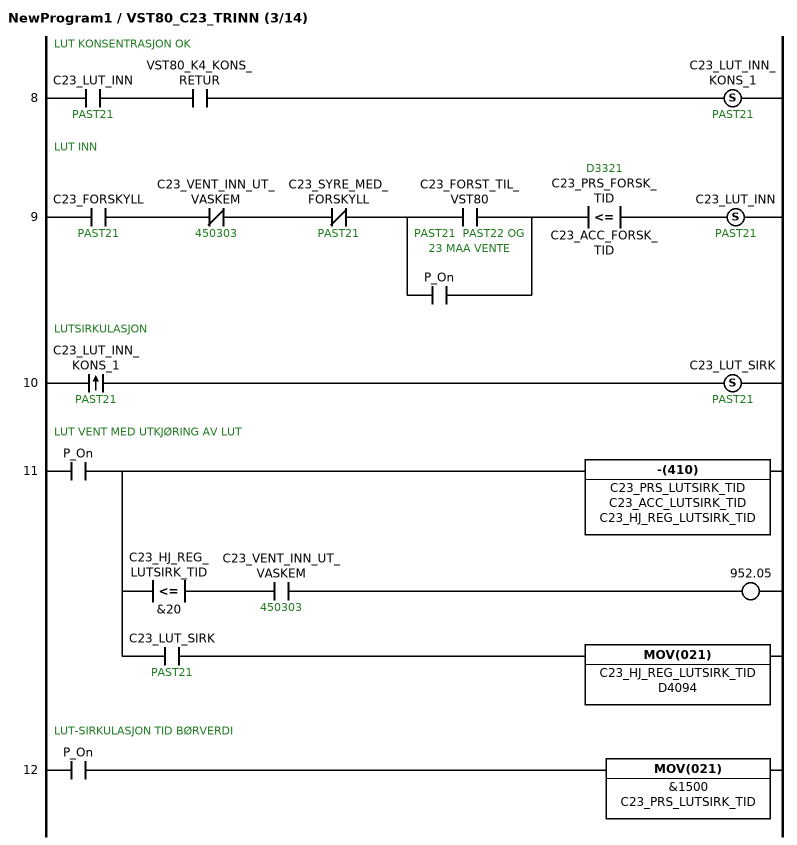
; [picture p408: NewProgram1 / VST80_C23_TRINN, rungs 8-12]
; rung 8: LUT KONSENTRASJON OK
LD C23_LUT_INN  ; PAST21
AND VST80_K4_KONS_RETUR
SET C23_LUT_INN_KONS_1  ; PAST21
; rung 9: LUT INN
LD C23_FORSKYLL  ; PAST21
ANDNOT C23_VENT_INN_UT_VASKEM  ; 450303
ANDNOT C23_SYRE_MED_FORSKYLL  ; PAST21
LD C23_FORST_TIL_VST80  ; PAST21  PAST22 OG 23 MAA VENTE
OR P_On
ANDLD
AND<=(315) C23_PRS_FORSK_TID C23_ACC_FORSK_TID  ; D3321
SET C23_LUT_INN  ; PAST21
; rung 10: LUTSIRKULASJON
@LD C23_LUT_INN_KONS_1  ; PAST21
SET C23_LUT_SIRK  ; PAST21
; rung 11: LUT VENT MED UTKJØRING AV LUT
LD P_On
OUT TR0
-(410) C23_PRS_LUTSIRK_TID C23_ACC_LUTSIRK_TID C23_HJ_REG_LUTSIRK_TID
AND<=(315) C23_HJ_REG_LUTSIRK_TID &20
AND C23_VENT_INN_UT_VASKEM  ; 450303
OUT 952.05
LD TR0
AND C23_LUT_SIRK  ; PAST21
MOV(021) C23_HJ_REG_LUTSIRK_TID D4094
; rung 12: LUT-SIRKULASJON TID BØRVERDI
LD P_On
MOV(021) &1500 C23_PRS_LUTSIRK_TID

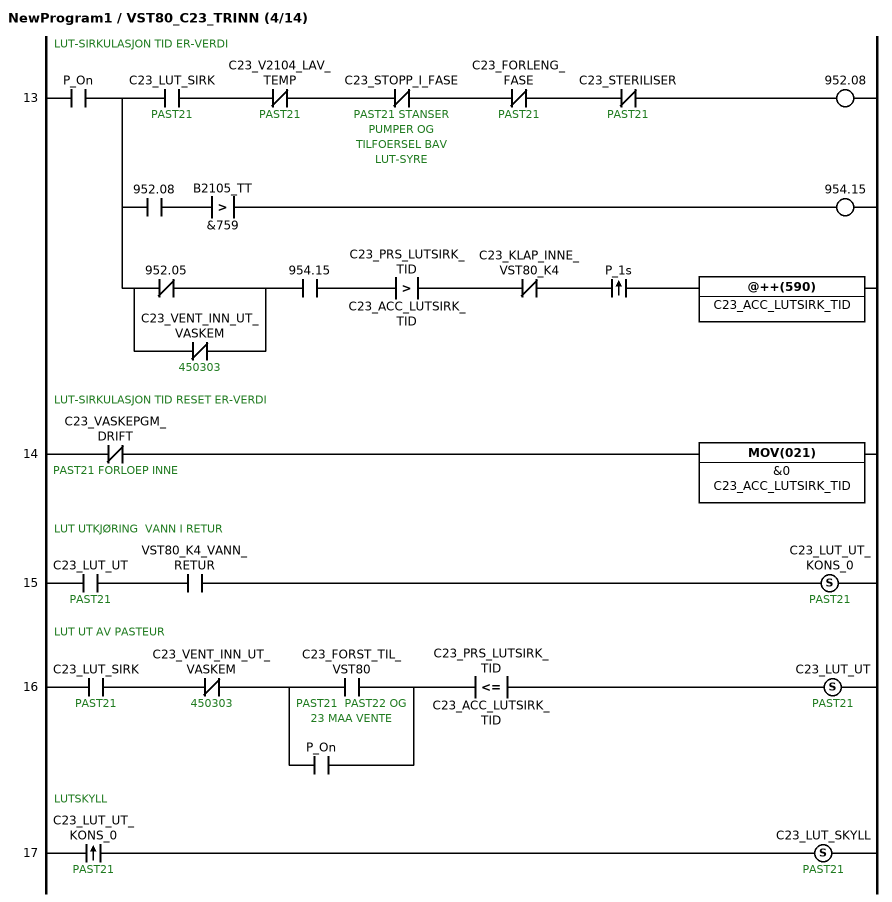
; rung 13: LUT-SIRKULASJON TID ER-VERDI
LD P_On
OUT TR0
AND C23_LUT_SIRK  ; PAST21
ANDNOT C23_V2104_LAV_TEMP  ; PAST21
ANDNOT C23_STOPP_I_FASE  ; PAST21 STANSER PUMPER OG TILFOERSEL BAV LUT-SYRE
ANDNOT C23_FORLENG_FASE  ; PAST21
ANDNOT C23_STERILISER  ; PAST21
OUT 952.08
LD TR0
AND 952.08
AND>(320) B2105_TT &759
OUT 954.15
LD TR0
LDNOT 952.05
ORNOT C23_VENT_INN_UT_VASKEM  ; 450303
ANDLD
AND 954.15
AND>(320) C23_PRS_LUTSIRK_TID C23_ACC_LUTSIRK_TID
ANDNOT C23_KLAP_INNE_VST80_K4
@AND P_1s
@++(590) C23_ACC_LUTSIRK_TID
; rung 14: LUT-SIRKULASJON TID RESET ER-VERDI
LDNOT C23_VASKEPGM_DRIFT  ; PAST21 FORLOEP INNE
MOV(021) &0 C23_ACC_LUTSIRK_TID
; rung 15: LUT UTKJØRING  VANN I RETUR
LD C23_LUT_UT  ; PAST21
AND VST80_K4_VANN_RETUR
SET C23_LUT_UT_KONS_0  ; PAST21
; rung 16: LUT UT AV PASTEUR
LD C23_LUT_SIRK  ; PAST21
ANDNOT C23_VENT_INN_UT_VASKEM  ; 450303
LD C23_FORST_TIL_VST80  ; PAST21  PAST22 OG 23 MAA VENTE
OR P_On
ANDLD
AND<=(315) C23_PRS_LUTSIRK_TID C23_ACC_LUTSIRK_TID
SET C23_LUT_UT  ; PAST21
; rung 17: LUTSKYLL
@LD C23_LUT_UT_KONS_0  ; PAST21
SET C23_LUT_SKYLL  ; PAST21

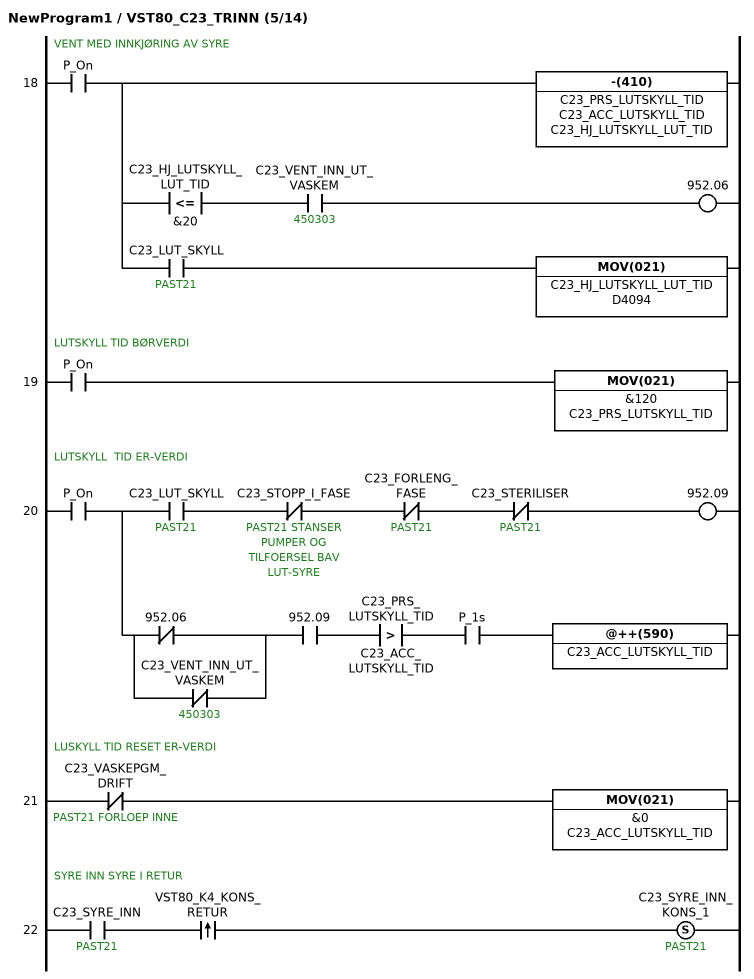
; rung 18: VENT MED INNKJØRING AV SYRE
LD P_On
OUT TR0
-(410) C23_PRS_LUTSKYLL_TID C23_ACC_LUTSKYLL_TID C23_HJ_LUTSKYLL_LUT_TID
AND<=(315) C23_HJ_LUTSKYLL_LUT_TID &20
AND C23_VENT_INN_UT_VASKEM  ; 450303
OUT 952.06
LD TR0
AND C23_LUT_SKYLL  ; PAST21
MOV(021) C23_HJ_LUTSKYLL_LUT_TID D4094
; rung 19: LUTSKYLL TID BØRVERDI
LD P_On
MOV(021) &120 C23_PRS_LUTSKYLL_TID
; rung 20: LUTSKYLL  TID ER-VERDI
LD P_On
OUT TR0
AND C23_LUT_SKYLL  ; PAST21
ANDNOT C23_STOPP_I_FASE  ; PAST21 STANSER PUMPER OG TILFOERSEL BAV LUT-SYRE
ANDNOT C23_FORLENG_FASE  ; PAST21
ANDNOT C23_STERILISER  ; PAST21
OUT 952.09
LD TR0
LDNOT 952.06
ORNOT C23_VENT_INN_UT_VASKEM  ; 450303
ANDLD
AND 952.09
AND>(320) C23_PRS_LUTSKYLL_TID C23_ACC_LUTSKYLL_TID
AND P_1s
@++(590) C23_ACC_LUTSKYLL_TID
; rung 21: LUSKYLL TID RESET ER-VERDI
LDNOT C23_VASKEPGM_DRIFT  ; PAST21 FORLOEP INNE
MOV(021) &0 C23_ACC_LUTSKYLL_TID
; rung 22: SYRE INN SYRE I RETUR
LD C23_SYRE_INN  ; PAST21
@AND VST80_K4_KONS_RETUR
SET C23_SYRE_INN_KONS_1  ; PAST21

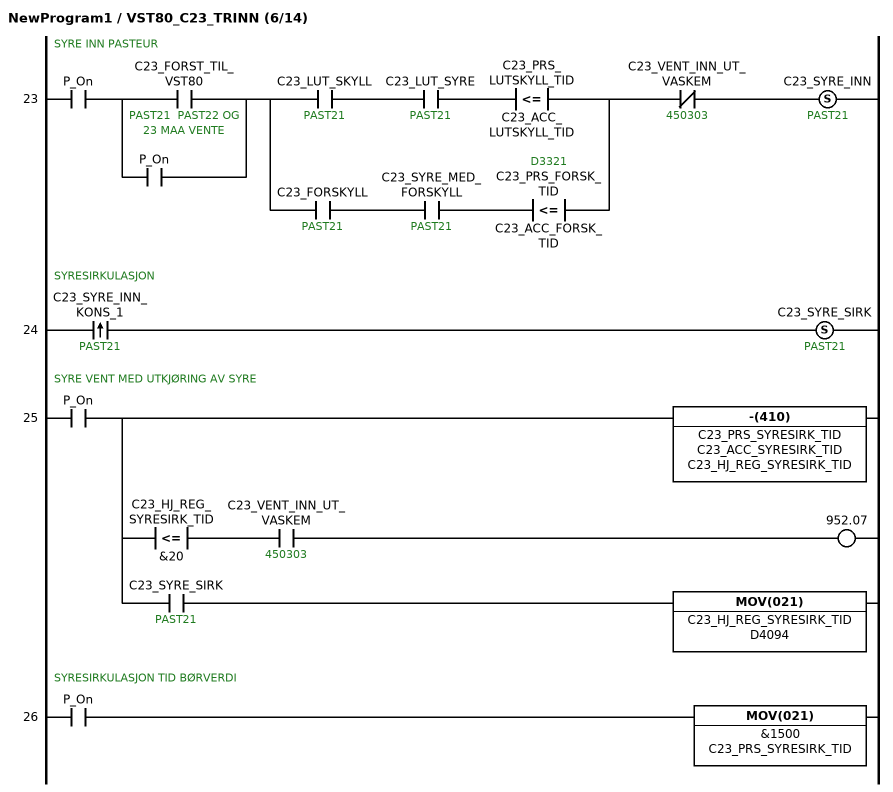
; rung 23: SYRE INN PASTEUR
LD P_On
LD C23_FORST_TIL_VST80  ; PAST21  PAST22 OG 23 MAA VENTE
OR P_On
ANDLD
LD C23_LUT_SKYLL  ; PAST21
AND C23_LUT_SYRE  ; PAST21
AND<=(315) C23_PRS_LUTSKYLL_TID C23_ACC_LUTSKYLL_TID
LD C23_FORSKYLL  ; PAST21
AND C23_SYRE_MED_FORSKYLL  ; PAST21
AND<=(315) C23_PRS_FORSK_TID C23_ACC_FORSK_TID  ; D3321
ORLD
ANDLD
ANDNOT C23_VENT_INN_UT_VASKEM  ; 450303
SET C23_SYRE_INN  ; PAST21
; rung 24: SYRESIRKULASJON
@LD C23_SYRE_INN_KONS_1  ; PAST21
SET C23_SYRE_SIRK  ; PAST21
; rung 25: SYRE VENT MED UTKJØRING AV SYRE
LD P_On
OUT TR0
-(410) C23_PRS_SYRESIRK_TID C23_ACC_SYRESIRK_TID C23_HJ_REG_SYRESIRK_TID
AND<=(315) C23_HJ_REG_SYRESIRK_TID &20
AND C23_VENT_INN_UT_VASKEM  ; 450303
OUT 952.07
LD TR0
AND C23_SYRE_SIRK  ; PAST21
MOV(021) C23_HJ_REG_SYRESIRK_TID D4094
; rung 26: SYRESIRKULASJON TID BØRVERDI
LD P_On
MOV(021) &1500 C23_PRS_SYRESIRK_TID

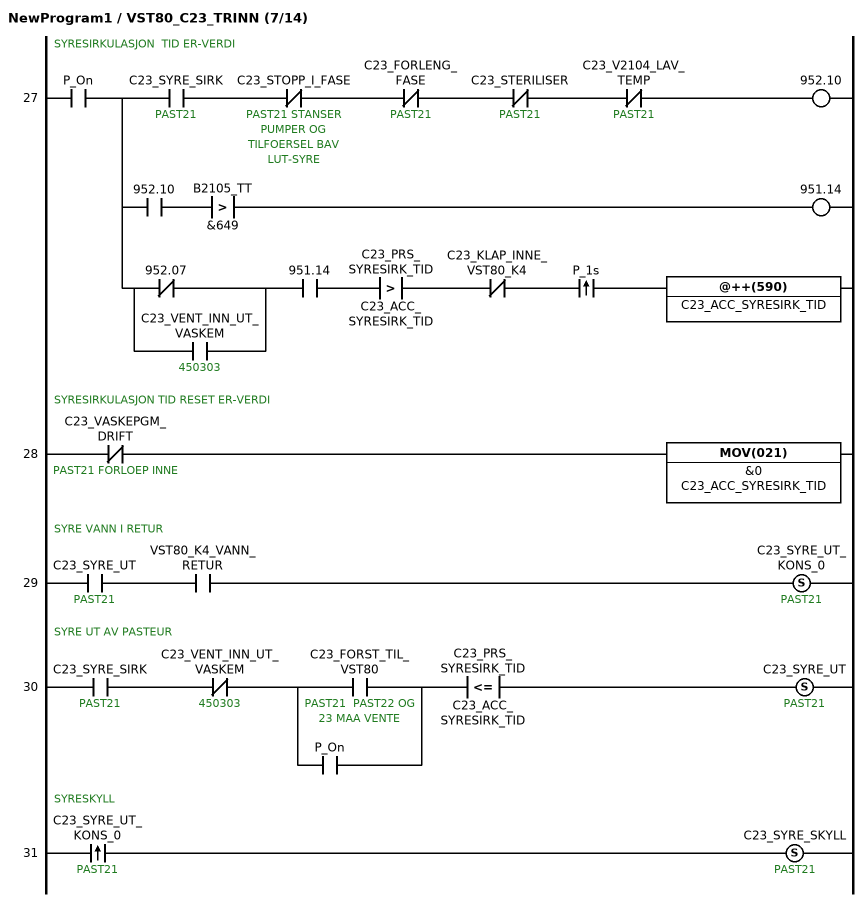
; rung 27: SYRESIRKULASJON  TID ER-VERDI
LD P_On
OUT TR0
AND C23_SYRE_SIRK  ; PAST21
ANDNOT C23_STOPP_I_FASE  ; PAST21 STANSER PUMPER OG TILFOERSEL BAV LUT-SYRE
ANDNOT C23_FORLENG_FASE  ; PAST21
ANDNOT C23_STERILISER  ; PAST21
ANDNOT C23_V2104_LAV_TEMP  ; PAST21
OUT 952.10
LD TR0
AND 952.10
AND>(320) B2105_TT &649
OUT 951.14
LD TR0
LDNOT 952.07
OR C23_VENT_INN_UT_VASKEM  ; 450303
ANDLD
AND 951.14
AND>(320) C23_PRS_SYRESIRK_TID C23_ACC_SYRESIRK_TID
ANDNOT C23_KLAP_INNE_VST80_K4
@AND P_1s
@++(590) C23_ACC_SYRESIRK_TID
; rung 28: SYRESIRKULASJON TID RESET ER-VERDI
LDNOT C23_VASKEPGM_DRIFT  ; PAST21 FORLOEP INNE
MOV(021) &0 C23_ACC_SYRESIRK_TID
; rung 29: SYRE VANN I RETUR
LD C23_SYRE_UT  ; PAST21
AND VST80_K4_VANN_RETUR
SET C23_SYRE_UT_KONS_0  ; PAST21
; rung 30: SYRE UT AV PASTEUR
LD C23_SYRE_SIRK  ; PAST21
ANDNOT C23_VENT_INN_UT_VASKEM  ; 450303
LD C23_FORST_TIL_VST80  ; PAST21  PAST22 OG 23 MAA VENTE
OR P_On
ANDLD
AND<=(315) C23_PRS_SYRESIRK_TID C23_ACC_SYRESIRK_TID
SET C23_SYRE_UT  ; PAST21
; rung 31: SYRESKYLL
@LD C23_SYRE_UT_KONS_0  ; PAST21
SET C23_SYRE_SKYLL  ; PAST21

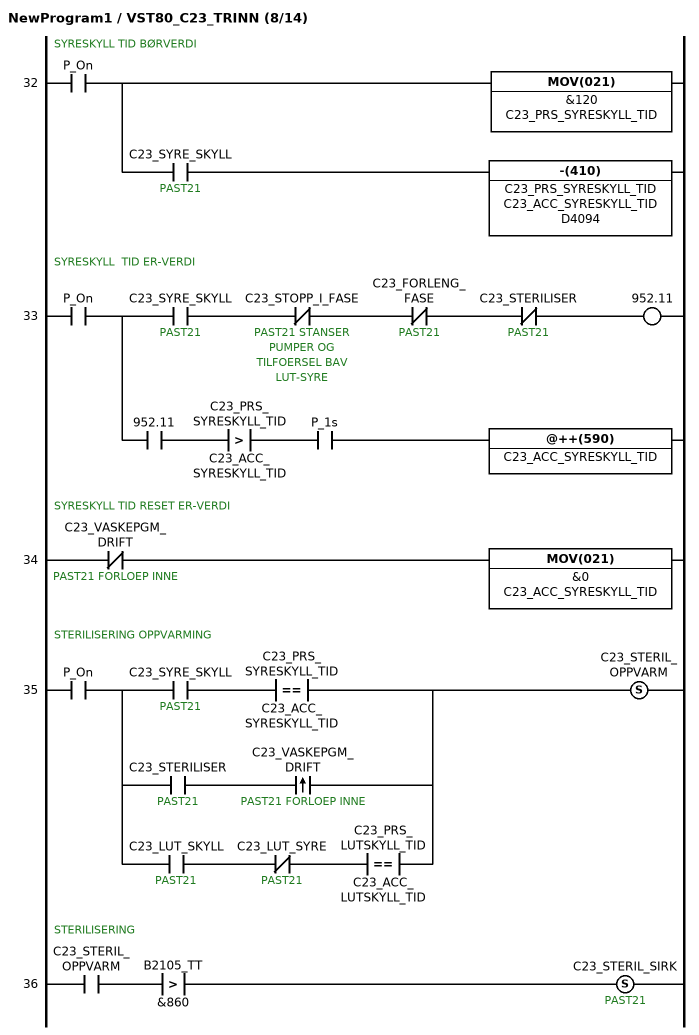
; rung 32: SYRESKYLL TID BØRVERDI
LD P_On
MOV(021) &120 C23_PRS_SYRESKYLL_TID
AND C23_SYRE_SKYLL  ; PAST21
-(410) C23_PRS_SYRESKYLL_TID C23_ACC_SYRESKYLL_TID D4094
; rung 33: SYRESKYLL  TID ER-VERDI
LD P_On
OUT TR0
AND C23_SYRE_SKYLL  ; PAST21
ANDNOT C23_STOPP_I_FASE  ; PAST21 STANSER PUMPER OG TILFOERSEL BAV LUT-SYRE
ANDNOT C23_FORLENG_FASE  ; PAST21
ANDNOT C23_STERILISER  ; PAST21
OUT 952.11
LD TR0
AND 952.11
AND>(320) C23_PRS_SYRESKYLL_TID C23_ACC_SYRESKYLL_TID
AND P_1s
@++(590) C23_ACC_SYRESKYLL_TID
; rung 34: SYRESKYLL TID RESET ER-VERDI
LDNOT C23_VASKEPGM_DRIFT  ; PAST21 FORLOEP INNE
MOV(021) &0 C23_ACC_SYRESKYLL_TID
; rung 35: STERILISERING OPPVARMING
LD P_On
LD C23_SYRE_SKYLL  ; PAST21
AND=(300) C23_PRS_SYRESKYLL_TID C23_ACC_SYRESKYLL_TID
LD C23_STERILISER  ; PAST21
@AND C23_VASKEPGM_DRIFT  ; PAST21 FORLOEP INNE
ORLD
LD C23_LUT_SKYLL  ; PAST21
ANDNOT C23_LUT_SYRE  ; PAST21
AND=(300) C23_PRS_LUTSKYLL_TID C23_ACC_LUTSKYLL_TID
ORLD
ANDLD
SET C23_STERIL_OPPVARM
; rung 36: STERILISERING
LD C23_STERIL_OPPVARM
AND>(320) B2105_TT &860
SET C23_STERIL_SIRK  ; PAST21

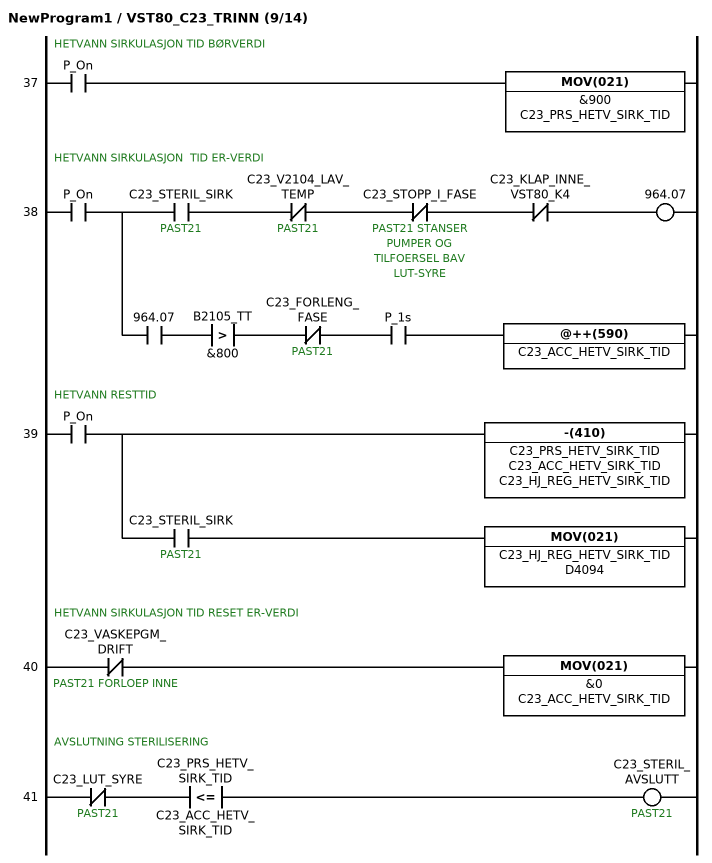
; rung 37: HETVANN SIRKULASJON TID BØRVERDI
LD P_On
MOV(021) &900 C23_PRS_HETV_SIRK_TID
; rung 38: HETVANN SIRKULASJON  TID ER-VERDI
LD P_On
OUT TR0
AND C23_STERIL_SIRK  ; PAST21
ANDNOT C23_V2104_LAV_TEMP  ; PAST21
ANDNOT C23_STOPP_I_FASE  ; PAST21 STANSER PUMPER OG TILFOERSEL BAV LUT-SYRE
ANDNOT C23_KLAP_INNE_VST80_K4
OUT 964.07
LD TR0
AND 964.07
AND>(320) B2105_TT &800
ANDNOT C23_FORLENG_FASE  ; PAST21
AND P_1s
@++(590) C23_ACC_HETV_SIRK_TID
; rung 39: HETVANN RESTTID
LD P_On
-(410) C23_PRS_HETV_SIRK_TID C23_ACC_HETV_SIRK_TID C23_HJ_REG_HETV_SIRK_TID
AND C23_STERIL_SIRK  ; PAST21
MOV(021) C23_HJ_REG_HETV_SIRK_TID D4094
; rung 40: HETVANN SIRKULASJON TID RESET ER-VERDI
LDNOT C23_VASKEPGM_DRIFT  ; PAST21 FORLOEP INNE
MOV(021) &0 C23_ACC_HETV_SIRK_TID
; rung 41: AVSLUTNING STERILISERING
LDNOT C23_LUT_SYRE  ; PAST21
AND<=(315) C23_PRS_HETV_SIRK_TID C23_ACC_HETV_SIRK_TID
OUT C23_STERIL_AVSLUTT  ; PAST21

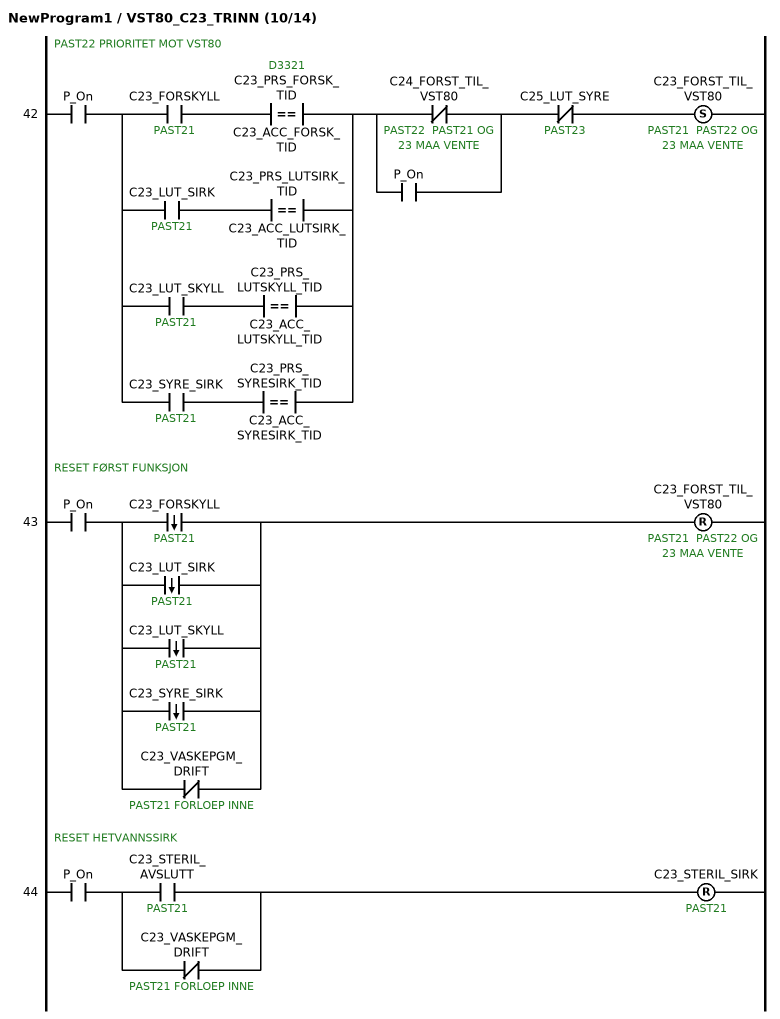
; rung 42: PAST22 PRIORITET MOT VST80
LD P_On
LD C23_FORSKYLL  ; PAST21
AND=(300) C23_PRS_FORSK_TID C23_ACC_FORSK_TID  ; D3321
LD C23_LUT_SIRK  ; PAST21
AND=(300) C23_PRS_LUTSIRK_TID C23_ACC_LUTSIRK_TID
ORLD
LD C23_LUT_SKYLL  ; PAST21
AND=(300) C23_PRS_LUTSKYLL_TID C23_ACC_LUTSKYLL_TID
ORLD
LD C23_SYRE_SIRK  ; PAST21
AND=(300) C23_PRS_SYRESIRK_TID C23_ACC_SYRESIRK_TID
ORLD
ANDLD
LDNOT C24_FORST_TIL_VST80  ; PAST22  PAST21 OG 23 MAA VENTE
OR P_On
ANDLD
ANDNOT C25_LUT_SYRE  ; PAST23
SET C23_FORST_TIL_VST80  ; PAST21  PAST22 OG 23 MAA VENTE
; rung 43: RESET FØRST FUNKSJON
LD P_On
%LD C23_FORSKYLL  ; PAST21
%OR C23_LUT_SIRK  ; PAST21
%OR C23_LUT_SKYLL  ; PAST21
%OR C23_SYRE_SIRK  ; PAST21
ORNOT C23_VASKEPGM_DRIFT  ; PAST21 FORLOEP INNE
ANDLD
RSET C23_FORST_TIL_VST80  ; PAST21  PAST22 OG 23 MAA VENTE
; rung 44: RESET HETVANNSSIRK
LD P_On
LD C23_STERIL_AVSLUTT  ; PAST21
ORNOT C23_VASKEPGM_DRIFT  ; PAST21 FORLOEP INNE
ANDLD
RSET C23_STERIL_SIRK  ; PAST21

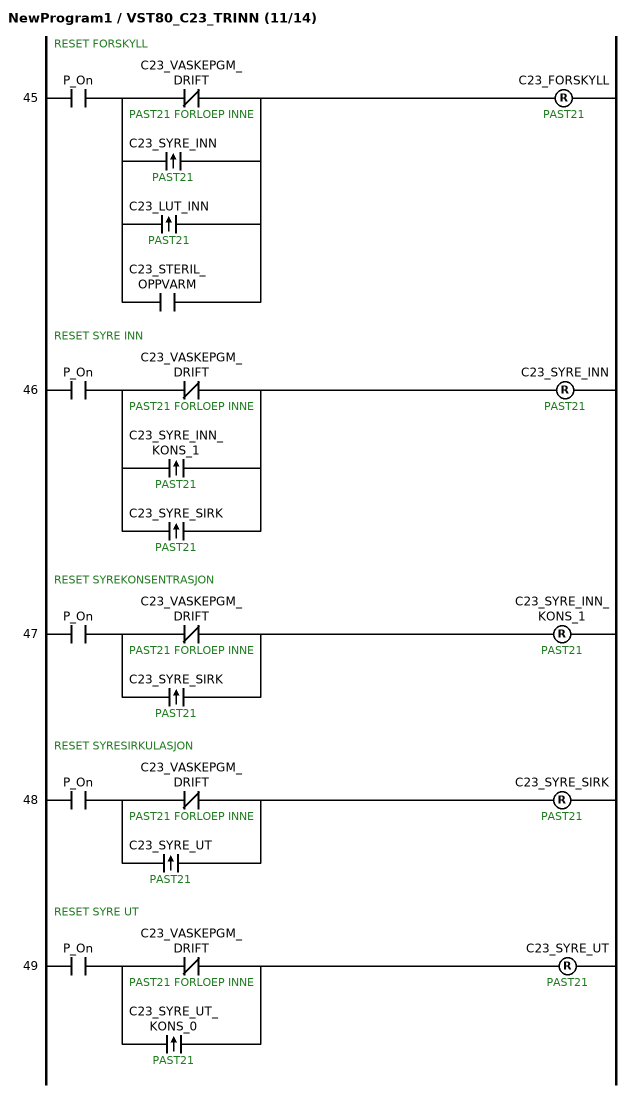
; rung 45: RESET FORSKYLL
LD P_On
LDNOT C23_VASKEPGM_DRIFT  ; PAST21 FORLOEP INNE
@OR C23_SYRE_INN  ; PAST21
@OR C23_LUT_INN  ; PAST21
OR C23_STERIL_OPPVARM
ANDLD
RSET C23_FORSKYLL  ; PAST21
; rung 46: RESET SYRE INN
LD P_On
LDNOT C23_VASKEPGM_DRIFT  ; PAST21 FORLOEP INNE
@OR C23_SYRE_INN_KONS_1  ; PAST21
@OR C23_SYRE_SIRK  ; PAST21
ANDLD
RSET C23_SYRE_INN  ; PAST21
; rung 47: RESET SYREKONSENTRASJON
LD P_On
LDNOT C23_VASKEPGM_DRIFT  ; PAST21 FORLOEP INNE
@OR C23_SYRE_SIRK  ; PAST21
ANDLD
RSET C23_SYRE_INN_KONS_1  ; PAST21
; rung 48: RESET SYRESIRKULASJON
LD P_On
LDNOT C23_VASKEPGM_DRIFT  ; PAST21 FORLOEP INNE
@OR C23_SYRE_UT  ; PAST21
ANDLD
RSET C23_SYRE_SIRK  ; PAST21
; rung 49: RESET SYRE UT
LD P_On
LDNOT C23_VASKEPGM_DRIFT  ; PAST21 FORLOEP INNE
@OR C23_SYRE_UT_KONS_0  ; PAST21
ANDLD
RSET C23_SYRE_UT  ; PAST21

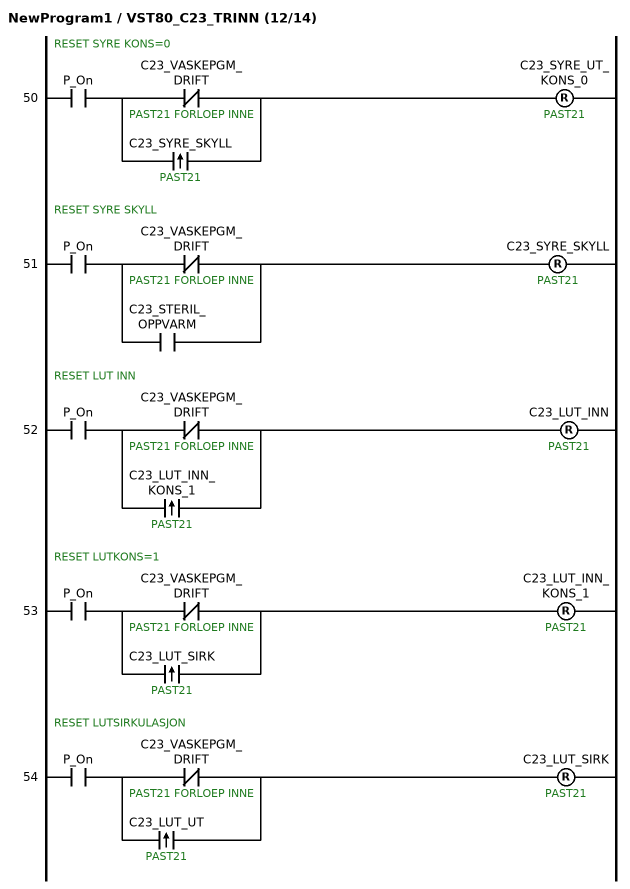
; rung 50: RESET SYRE KONS=0
LD P_On
LDNOT C23_VASKEPGM_DRIFT  ; PAST21 FORLOEP INNE
@OR C23_SYRE_SKYLL  ; PAST21
ANDLD
RSET C23_SYRE_UT_KONS_0  ; PAST21
; rung 51: RESET SYRE SKYLL
LD P_On
LDNOT C23_VASKEPGM_DRIFT  ; PAST21 FORLOEP INNE
OR C23_STERIL_OPPVARM
ANDLD
RSET C23_SYRE_SKYLL  ; PAST21
; rung 52: RESET LUT INN
LD P_On
LDNOT C23_VASKEPGM_DRIFT  ; PAST21 FORLOEP INNE
@OR C23_LUT_INN_KONS_1  ; PAST21
ANDLD
RSET C23_LUT_INN  ; PAST21
; rung 53: RESET LUTKONS=1
LD P_On
LDNOT C23_VASKEPGM_DRIFT  ; PAST21 FORLOEP INNE
@OR C23_LUT_SIRK  ; PAST21
ANDLD
RSET C23_LUT_INN_KONS_1  ; PAST21
; rung 54: RESET LUTSIRKULASJON
LD P_On
LDNOT C23_VASKEPGM_DRIFT  ; PAST21 FORLOEP INNE
@OR C23_LUT_UT  ; PAST21
ANDLD
RSET C23_LUT_SIRK  ; PAST21

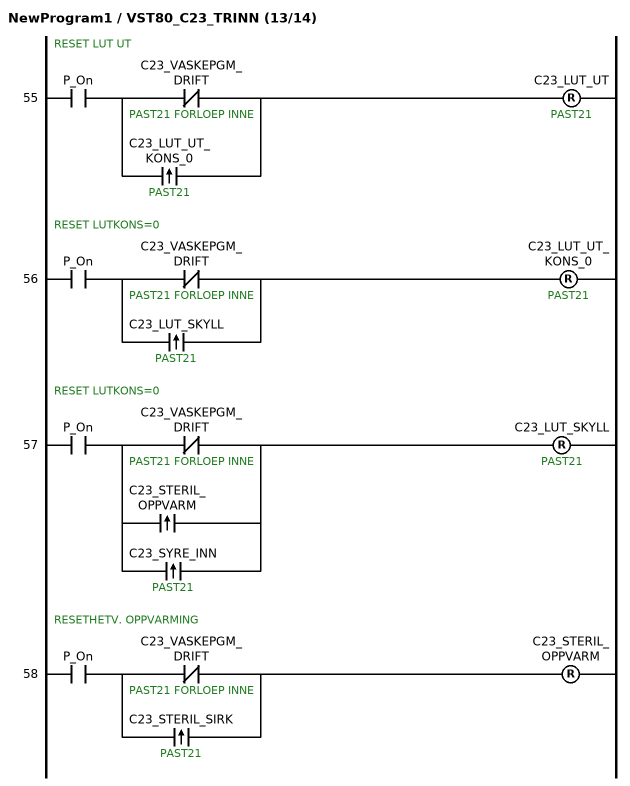
; rung 55: RESET LUT UT
LD P_On
LDNOT C23_VASKEPGM_DRIFT  ; PAST21 FORLOEP INNE
@OR C23_LUT_UT_KONS_0  ; PAST21
ANDLD
RSET C23_LUT_UT  ; PAST21
; rung 56: RESET LUTKONS=0
LD P_On
LDNOT C23_VASKEPGM_DRIFT  ; PAST21 FORLOEP INNE
@OR C23_LUT_SKYLL  ; PAST21
ANDLD
RSET C23_LUT_UT_KONS_0  ; PAST21
; rung 57: RESET LUTKONS=0
LD P_On
LDNOT C23_VASKEPGM_DRIFT  ; PAST21 FORLOEP INNE
@OR C23_STERIL_OPPVARM
@OR C23_SYRE_INN  ; PAST21
ANDLD
RSET C23_LUT_SKYLL  ; PAST21
; rung 58: RESETHETV. OPPVARMING
LD P_On
LDNOT C23_VASKEPGM_DRIFT  ; PAST21 FORLOEP INNE
@OR C23_STERIL_SIRK  ; PAST21
ANDLD
RSET C23_STERIL_OPPVARM

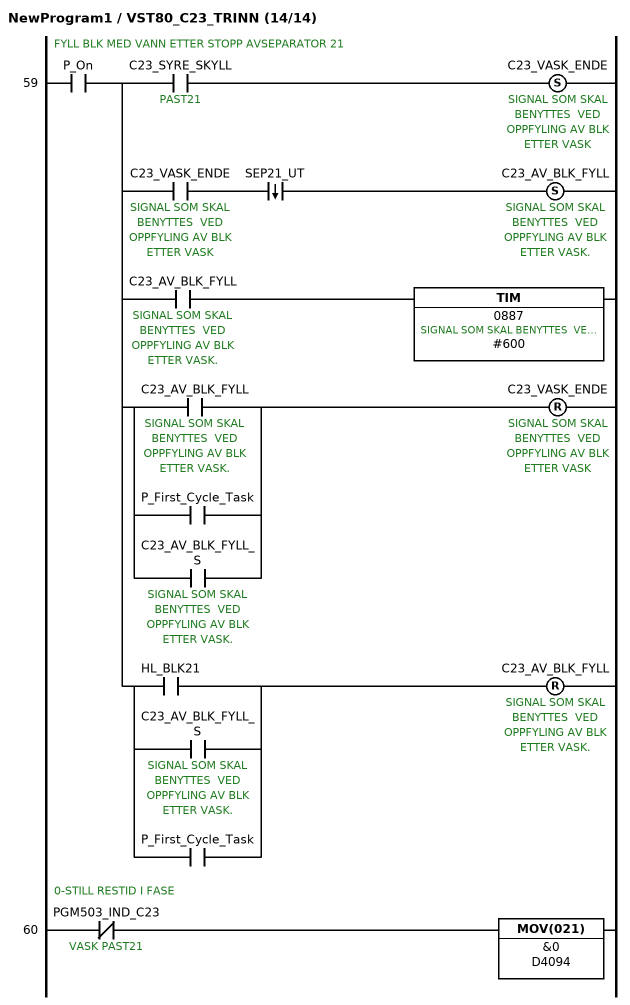
; rung 59: FYLL BLK MED VANN ETTER STOPP AVSEPARATOR 21
LD P_On
OUT TR0
AND C23_SYRE_SKYLL  ; PAST21
SET C23_VASK_ENDE  ; SIGNAL SOM SKAL BENYTTES  VED OPPFYLING AV BLK ETTER VASK
LD TR0
AND C23_VASK_ENDE  ; SIGNAL SOM SKAL BENYTTES  VED OPPFYLING AV BLK ETTER VASK
%AND SEP21_UT
SET C23_AV_BLK_FYLL  ; SIGNAL SOM SKAL BENYTTES  VED OPPFYLING AV BLK ETTER VASK.
LD TR0
AND C23_AV_BLK_FYLL  ; SIGNAL SOM SKAL BENYTTES  VED OPPFYLING AV BLK ETTER VASK.
TIM 0887 #600  ; SIGNAL SOM SKAL BENYTTES  VED OPPFYLING AV BLK ETTER VASK.
LD TR0
LD C23_AV_BLK_FYLL  ; SIGNAL SOM SKAL BENYTTES  VED OPPFYLING AV BLK ETTER VASK.
OR P_First_Cycle_Task
OR C23_AV_BLK_FYLL_S  ; SIGNAL SOM SKAL BENYTTES  VED OPPFYLING AV BLK ETTER VASK.
ANDLD
RSET C23_VASK_ENDE  ; SIGNAL SOM SKAL BENYTTES  VED OPPFYLING AV BLK ETTER VASK
LD TR0
LD HL_BLK21
OR C23_AV_BLK_FYLL_S  ; SIGNAL SOM SKAL BENYTTES  VED OPPFYLING AV BLK ETTER VASK.
OR P_First_Cycle_Task
ANDLD
RSET C23_AV_BLK_FYLL  ; SIGNAL SOM SKAL BENYTTES  VED OPPFYLING AV BLK ETTER VASK.
; rung 60: 0-STILL RESTID I FASE
LDNOT PGM503_IND_C23  ; VASK PAST21
MOV(021) &0 D4094

### Section VST80_C23_GRAFIKK_TEKSTER

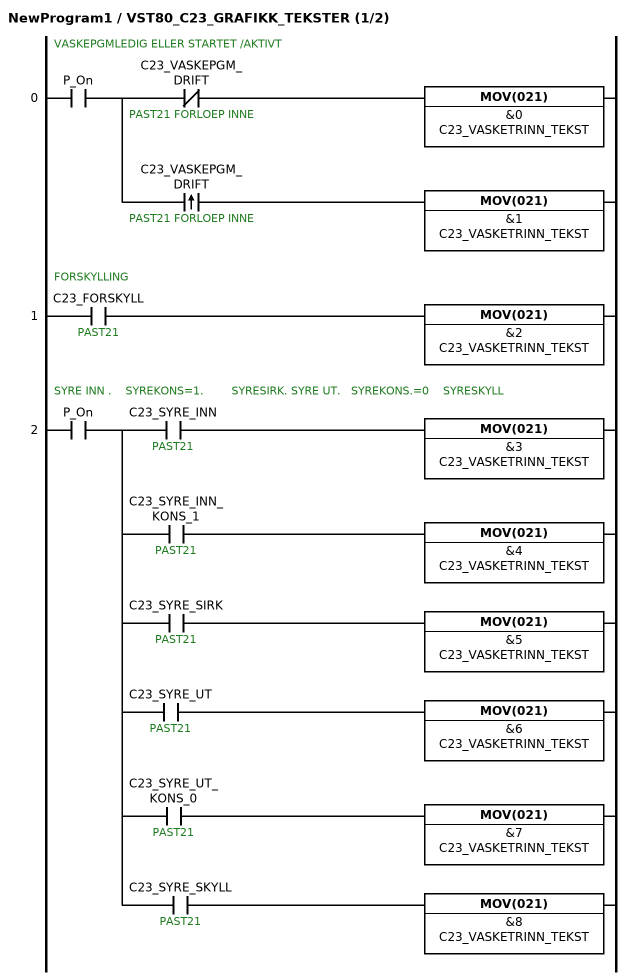
; rung 0: VASKEPGMLEDIG ELLER STARTET /AKTIVT
LD P_On
OUT TR0
ANDNOT C23_VASKEPGM_DRIFT  ; PAST21 FORLOEP INNE
MOV(021) &0 C23_VASKETRINN_TEKST
LD TR0
@AND C23_VASKEPGM_DRIFT  ; PAST21 FORLOEP INNE
MOV(021) &1 C23_VASKETRINN_TEKST
; rung 1: FORSKYLLING
LD C23_FORSKYLL  ; PAST21
MOV(021) &2 C23_VASKETRINN_TEKST
; rung 2: SYRE INN .    SYREKONS=1.        SYRESIRK. SYRE UT.   SYREKONS.=0    SYRESKYLL
LD P_On
OUT TR0
AND C23_SYRE_INN  ; PAST21
MOV(021) &3 C23_VASKETRINN_TEKST
LD TR0
AND C23_SYRE_INN_KONS_1  ; PAST21
MOV(021) &4 C23_VASKETRINN_TEKST
LD TR0
AND C23_SYRE_SIRK  ; PAST21
MOV(021) &5 C23_VASKETRINN_TEKST
LD TR0
AND C23_SYRE_UT  ; PAST21
MOV(021) &6 C23_VASKETRINN_TEKST
LD TR0
AND C23_SYRE_UT_KONS_0  ; PAST21
MOV(021) &7 C23_VASKETRINN_TEKST
LD TR0
AND C23_SYRE_SKYLL  ; PAST21
MOV(021) &8 C23_VASKETRINN_TEKST

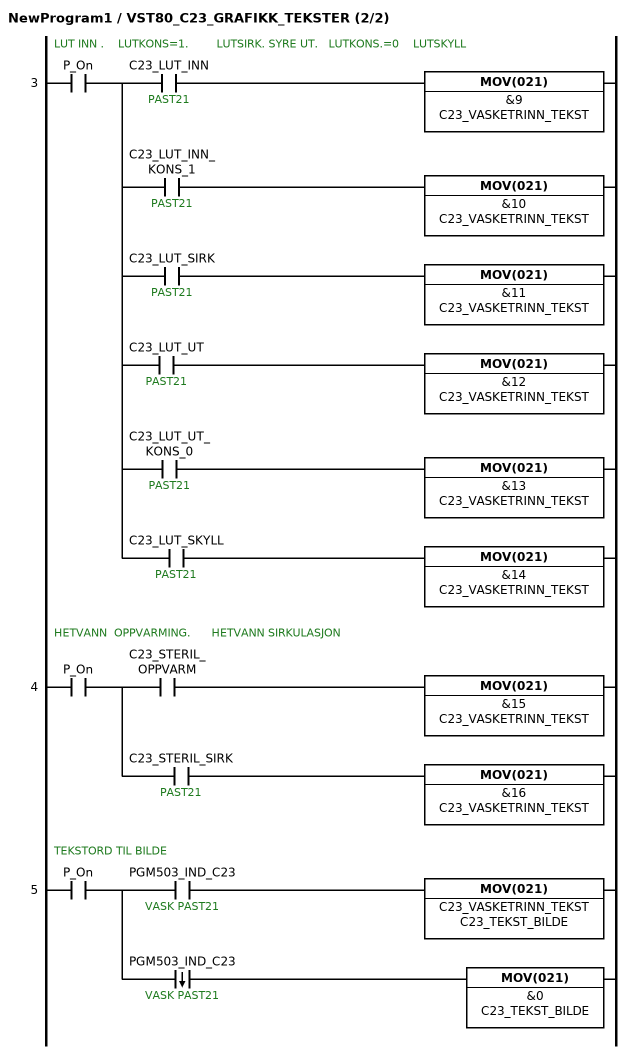
; rung 3: LUT INN .    LUTKONS=1.        LUTSIRK. SYRE UT.   LUTKONS.=0    LUTSKYLL
LD P_On
OUT TR0
AND C23_LUT_INN  ; PAST21
MOV(021) &9 C23_VASKETRINN_TEKST
LD TR0
AND C23_LUT_INN_KONS_1  ; PAST21
MOV(021) &10 C23_VASKETRINN_TEKST
LD TR0
AND C23_LUT_SIRK  ; PAST21
MOV(021) &11 C23_VASKETRINN_TEKST
LD TR0
AND C23_LUT_UT  ; PAST21
MOV(021) &12 C23_VASKETRINN_TEKST
LD TR0
AND C23_LUT_UT_KONS_0  ; PAST21
MOV(021) &13 C23_VASKETRINN_TEKST
LD TR0
AND C23_LUT_SKYLL  ; PAST21
MOV(021) &14 C23_VASKETRINN_TEKST
; rung 4: HETVANN  OPPVARMING.      HETVANN SIRKULASJON
LD P_On
OUT TR0
AND C23_STERIL_OPPVARM
MOV(021) &15 C23_VASKETRINN_TEKST
LD TR0
AND C23_STERIL_SIRK  ; PAST21
MOV(021) &16 C23_VASKETRINN_TEKST
; rung 5: TEKSTORD TIL BILDE
LD P_On
OUT TR0
AND PGM503_IND_C23  ; VASK PAST21
MOV(021) C23_VASKETRINN_TEKST C23_TEKST_BILDE
LD TR0
%AND PGM503_IND_C23  ; VASK PAST21
MOV(021) &0 C23_TEKST_BILDE

### Section C23_VASKERAPPORT

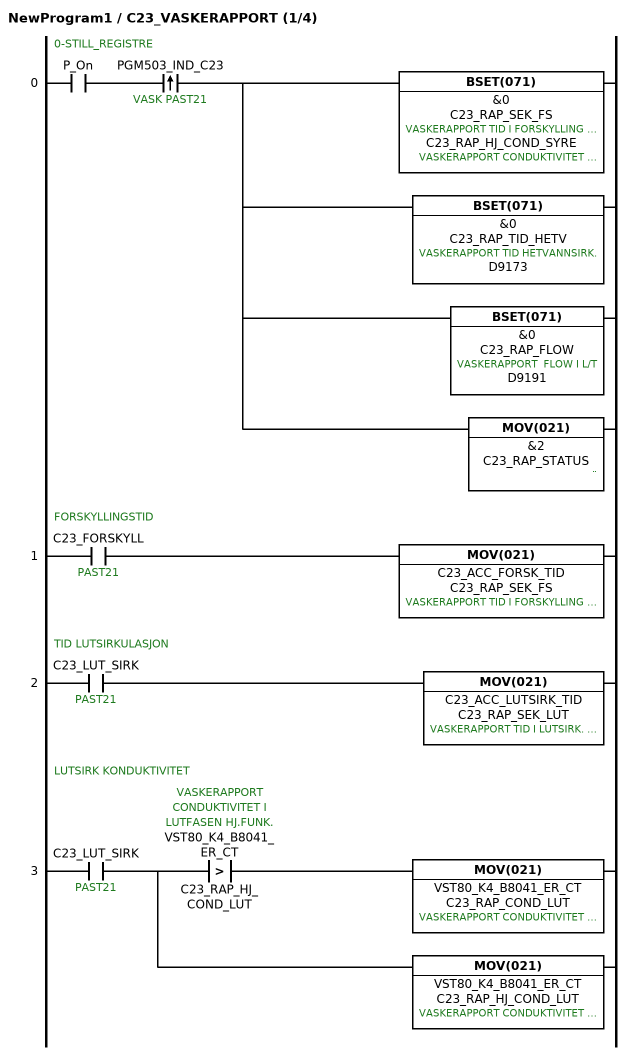
; rung 0: 0-STILL_REGISTRE
LD P_On
@AND PGM503_IND_C23  ; VASK PAST21
BSET(071) &0 C23_RAP_SEK_FS C23_RAP_HJ_COND_SYRE  ; VASKERAPPORT TID I FORSKYLLING I SEKUNDER, VASKERAPPORT CONDUKTIVITET I SYREFASEN HJ.FUNK.
BSET(071) &0 C23_RAP_TID_HETV D9173  ; VASKERAPPORT TID HETVANNSIRK.
BSET(071) &0 C23_RAP_FLOW D9191  ; VASKERAPPORT  FLOW I L/T
MOV(021) &2 C23_RAP_STATUS  ; ¨
; rung 1: FORSKYLLINGSTID
LD C23_FORSKYLL  ; PAST21
MOV(021) C23_ACC_FORSK_TID C23_RAP_SEK_FS  ; VASKERAPPORT TID I FORSKYLLING I SEKUNDER
; rung 2: TID LUTSIRKULASJON
LD C23_LUT_SIRK  ; PAST21
MOV(021) C23_ACC_LUTSIRK_TID C23_RAP_SEK_LUT  ; VASKERAPPORT TID I LUTSIRK. I SEKUNDER
; rung 3: LUTSIRK KONDUKTIVITET
LD C23_LUT_SIRK  ; PAST21
OUT TR0
AND>(320) VST80_K4_B8041_ER_CT C23_RAP_HJ_COND_LUT  ; VASKERAPPORT CONDUKTIVITET I LUTFASEN HJ.FUNK.
MOV(021) VST80_K4_B8041_ER_CT C23_RAP_COND_LUT  ; VASKERAPPORT CONDUKTIVITET I LUTFASEN
LD TR0
MOV(021) VST80_K4_B8041_ER_CT C23_RAP_HJ_COND_LUT  ; VASKERAPPORT CONDUKTIVITET I LUTFASEN HJ.FUNK.

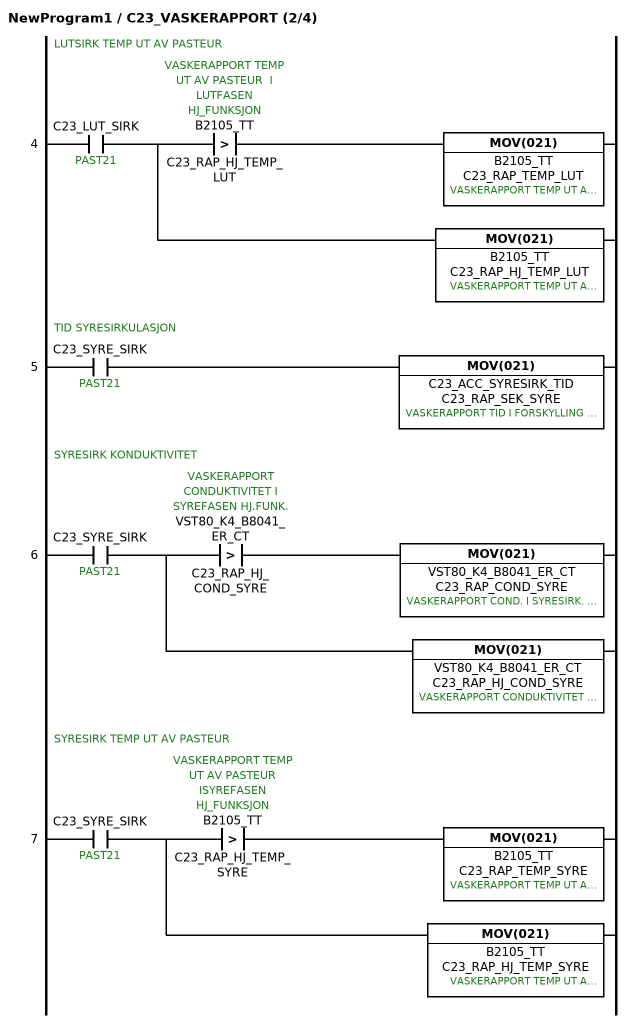
; rung 4: LUTSIRK TEMP UT AV PASTEUR
LD C23_LUT_SIRK  ; PAST21
OUT TR0
AND>(320) B2105_TT C23_RAP_HJ_TEMP_LUT  ; VASKERAPPORT TEMP UT AV PASTEUR  I LUTFASEN HJ_FUNKSJON
MOV(021) B2105_TT C23_RAP_TEMP_LUT  ; VASKERAPPORT TEMP UT AV PASTEUR  I LUTFASEN
LD TR0
MOV(021) B2105_TT C23_RAP_HJ_TEMP_LUT  ; VASKERAPPORT TEMP UT AV PASTEUR  I LUTFASEN HJ_FUNKSJON
; rung 5: TID SYRESIRKULASJON
LD C23_SYRE_SIRK  ; PAST21
MOV(021) C23_ACC_SYRESIRK_TID C23_RAP_SEK_SYRE  ; VASKERAPPORT TID I FORSKYLLING I SEKUNDER
; rung 6: SYRESIRK KONDUKTIVITET
LD C23_SYRE_SIRK  ; PAST21
OUT TR0
AND>(320) VST80_K4_B8041_ER_CT C23_RAP_HJ_COND_SYRE  ; VASKERAPPORT CONDUKTIVITET I SYREFASEN HJ.FUNK.
MOV(021) VST80_K4_B8041_ER_CT C23_RAP_COND_SYRE  ; VASKERAPPORT COND. I SYRESIRK. I SEKUNDER
LD TR0
MOV(021) VST80_K4_B8041_ER_CT C23_RAP_HJ_COND_SYRE  ; VASKERAPPORT CONDUKTIVITET I SYREFASEN HJ.FUNK.
; rung 7: SYRESIRK TEMP UT AV PASTEUR
LD C23_SYRE_SIRK  ; PAST21
OUT TR0
AND>(320) B2105_TT C23_RAP_HJ_TEMP_SYRE  ; VASKERAPPORT TEMP UT AV PASTEUR ISYREFASEN HJ_FUNKSJON
MOV(021) B2105_TT C23_RAP_TEMP_SYRE  ; VASKERAPPORT TEMP UT AV PASTEUR ISYREFASEN
LD TR0
MOV(021) B2105_TT C23_RAP_HJ_TEMP_SYRE  ; VASKERAPPORT TEMP UT AV PASTEUR ISYREFASEN HJ_FUNKSJON

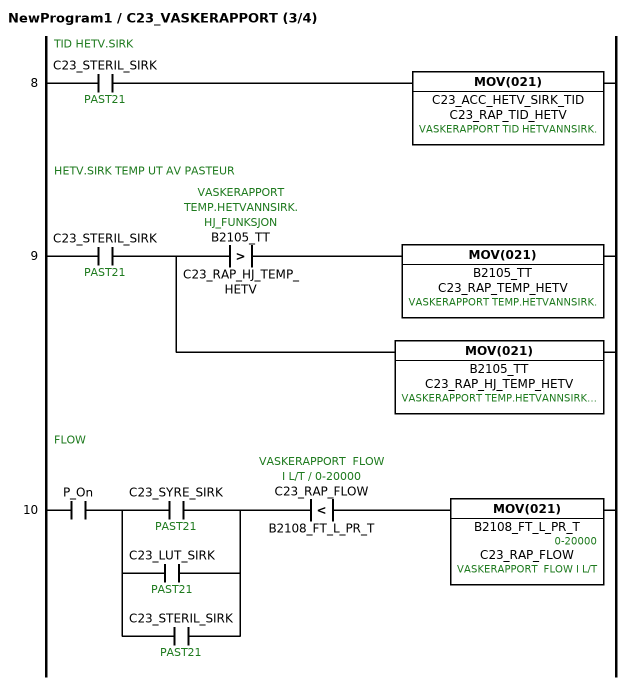
; rung 8: TID HETV.SIRK
LD C23_STERIL_SIRK  ; PAST21
MOV(021) C23_ACC_HETV_SIRK_TID C23_RAP_TID_HETV  ; VASKERAPPORT TID HETVANNSIRK.
; rung 9: HETV.SIRK TEMP UT AV PASTEUR
LD C23_STERIL_SIRK  ; PAST21
OUT TR0
AND>(320) B2105_TT C23_RAP_HJ_TEMP_HETV  ; VASKERAPPORT TEMP.HETVANNSIRK. HJ_FUNKSJON
MOV(021) B2105_TT C23_RAP_TEMP_HETV  ; VASKERAPPORT TEMP.HETVANNSIRK.
LD TR0
MOV(021) B2105_TT C23_RAP_HJ_TEMP_HETV  ; VASKERAPPORT TEMP.HETVANNSIRK. HJ_FUNKSJON
; rung 10: FLOW
LD P_On
LD C23_SYRE_SIRK  ; PAST21
OR C23_LUT_SIRK  ; PAST21
OR C23_STERIL_SIRK  ; PAST21
ANDLD
AND<(310) C23_RAP_FLOW B2108_FT_L_PR_T  ; VASKERAPPORT  FLOW I L/T, 0-20000
MOV(021) B2108_FT_L_PR_T C23_RAP_FLOW  ; 0-20000, VASKERAPPORT  FLOW I L/T

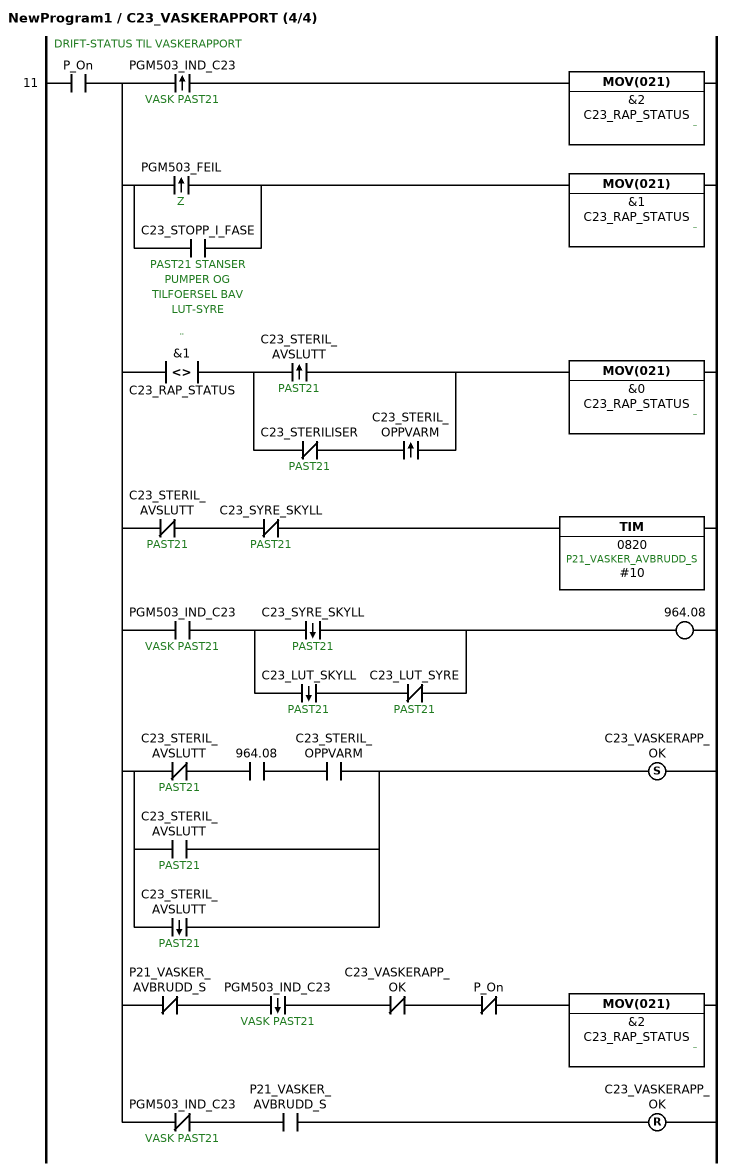
; rung 11: DRIFT-STATUS TIL VASKERAPPORT
LD P_On
OUT TR0
@AND PGM503_IND_C23  ; VASK PAST21
MOV(021) &2 C23_RAP_STATUS  ; ¨
LD TR0
@LD PGM503_FEIL  ; Z
OR C23_STOPP_I_FASE  ; PAST21 STANSER PUMPER OG TILFOERSEL BAV LUT-SYRE
ANDLD
MOV(021) &1 C23_RAP_STATUS  ; ¨
LD TR0
AND<>(305) &1 C23_RAP_STATUS  ; ¨
@LD C23_STERIL_AVSLUTT  ; PAST21
LDNOT C23_STERILISER  ; PAST21
@AND C23_STERIL_OPPVARM
ORLD
ANDLD
MOV(021) &0 C23_RAP_STATUS  ; ¨
LD TR0
ANDNOT C23_STERIL_AVSLUTT  ; PAST21
ANDNOT C23_SYRE_SKYLL  ; PAST21
TIM 0820 #10  ; P21_VASKER_AVBRUDD_S
LD TR0
AND PGM503_IND_C23  ; VASK PAST21
%LD C23_SYRE_SKYLL  ; PAST21
%LD C23_LUT_SKYLL  ; PAST21
ANDNOT C23_LUT_SYRE  ; PAST21
ORLD
ANDLD
OUT 964.08
LD TR0
LDNOT C23_STERIL_AVSLUTT  ; PAST21
AND 964.08
AND C23_STERIL_OPPVARM
OR C23_STERIL_AVSLUTT  ; PAST21
%OR C23_STERIL_AVSLUTT  ; PAST21
ANDLD
SET C23_VASKERAPP_OK
LD TR0
ANDNOT P21_VASKER_AVBRUDD_S
%AND PGM503_IND_C23  ; VASK PAST21
ANDNOT C23_VASKERAPP_OK
ANDNOT P_On
MOV(021) &2 C23_RAP_STATUS  ; ¨
LD TR0
ANDNOT PGM503_IND_C23  ; VASK PAST21
AND P21_VASKER_AVBRUDD_S
RSET C23_VASKERAPP_OK

### Section C24_FUNKSJONER

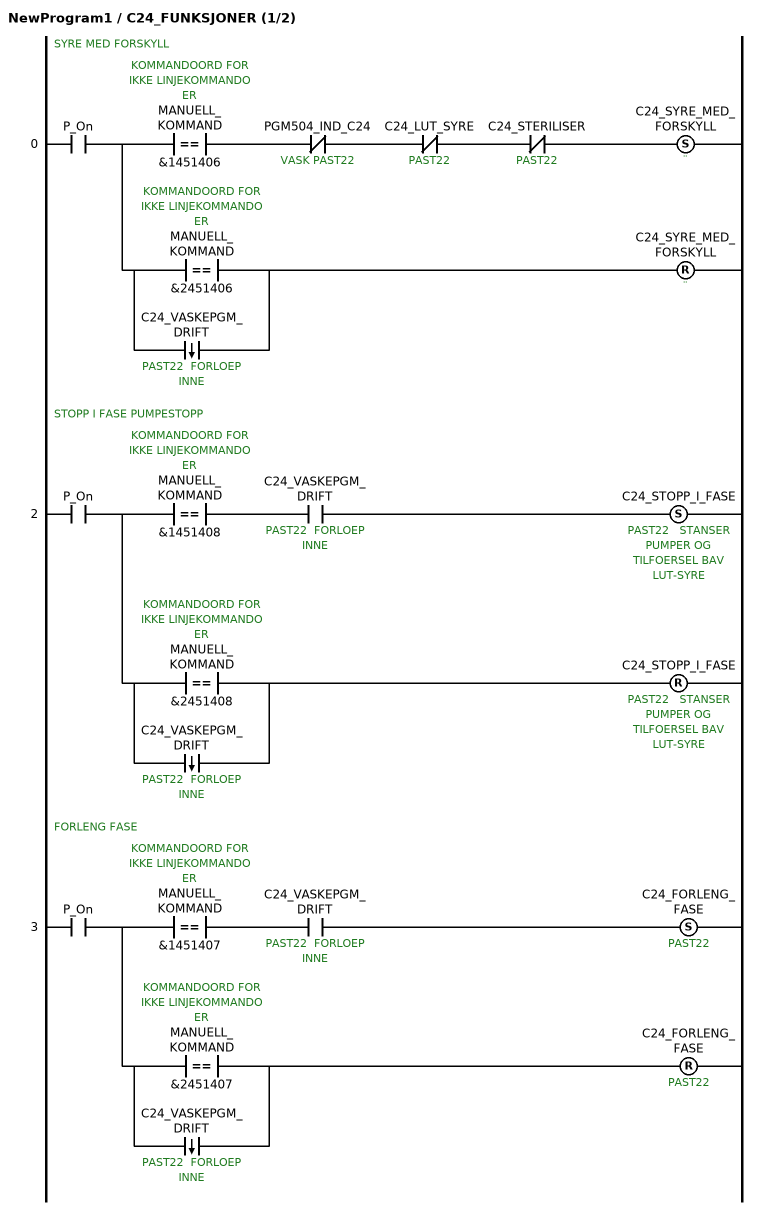
; rung 0: SYRE MED FORSKYLL
LD P_On
OUT TR0
AND=L(301) MANUELL_KOMMAND &1451406  ; KOMMANDOORD FOR IKKE LINJEKOMMANDOER
ANDNOT PGM504_IND_C24  ; VASK PAST22
ANDNOT C24_LUT_SYRE  ; PAST22
ANDNOT C24_STERILISER  ; PAST22
SET C24_SYRE_MED_FORSKYLL  ; ¨
LD TR0
LD=L(301) MANUELL_KOMMAND &2451406  ; KOMMANDOORD FOR IKKE LINJEKOMMANDOER
%OR C24_VASKEPGM_DRIFT  ; PAST22  FORLOEP INNE
ANDLD
RSET C24_SYRE_MED_FORSKYLL  ; ¨
; rung 1: STOPP ETTER VASKEMIDDEL
; rung 2: STOPP I FASE PUMPESTOPP
LD P_On
OUT TR0
AND=L(301) MANUELL_KOMMAND &1451408  ; KOMMANDOORD FOR IKKE LINJEKOMMANDOER
AND C24_VASKEPGM_DRIFT  ; PAST22  FORLOEP INNE
SET C24_STOPP_I_FASE  ; PAST22   STANSER PUMPER OG TILFOERSEL BAV LUT-SYRE
LD TR0
LD=L(301) MANUELL_KOMMAND &2451408  ; KOMMANDOORD FOR IKKE LINJEKOMMANDOER
%OR C24_VASKEPGM_DRIFT  ; PAST22  FORLOEP INNE
ANDLD
RSET C24_STOPP_I_FASE  ; PAST22   STANSER PUMPER OG TILFOERSEL BAV LUT-SYRE
; rung 3: FORLENG FASE
LD P_On
OUT TR0
AND=L(301) MANUELL_KOMMAND &1451407  ; KOMMANDOORD FOR IKKE LINJEKOMMANDOER
AND C24_VASKEPGM_DRIFT  ; PAST22  FORLOEP INNE
SET C24_FORLENG_FASE  ; PAST22
LD TR0
LD=L(301) MANUELL_KOMMAND &2451407  ; KOMMANDOORD FOR IKKE LINJEKOMMANDOER
%OR C24_VASKEPGM_DRIFT  ; PAST22  FORLOEP INNE
ANDLD
RSET C24_FORLENG_FASE  ; PAST22

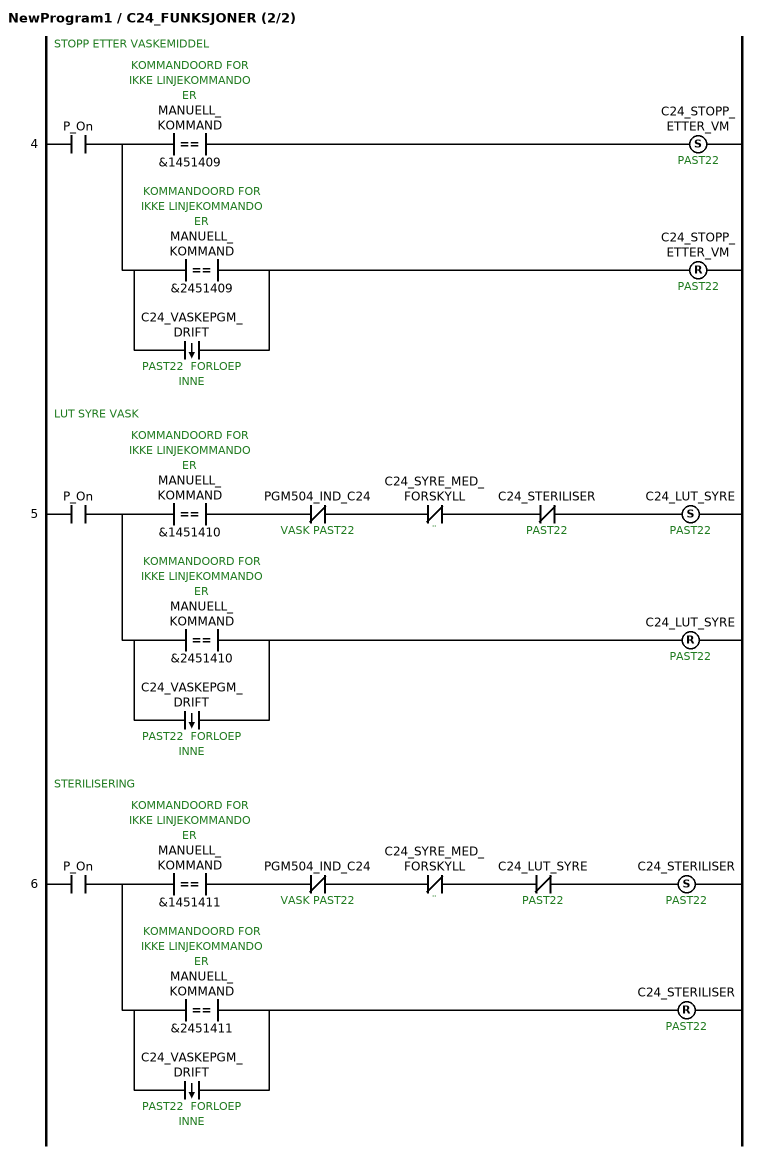
; rung 4: STOPP ETTER VASKEMIDDEL
LD P_On
OUT TR0
AND=L(301) MANUELL_KOMMAND &1451409  ; KOMMANDOORD FOR IKKE LINJEKOMMANDOER
SET C24_STOPP_ETTER_VM  ; PAST22
LD TR0
LD=L(301) MANUELL_KOMMAND &2451409  ; KOMMANDOORD FOR IKKE LINJEKOMMANDOER
%OR C24_VASKEPGM_DRIFT  ; PAST22  FORLOEP INNE
ANDLD
RSET C24_STOPP_ETTER_VM  ; PAST22
; rung 5: LUT SYRE VASK
LD P_On
OUT TR0
AND=L(301) MANUELL_KOMMAND &1451410  ; KOMMANDOORD FOR IKKE LINJEKOMMANDOER
ANDNOT PGM504_IND_C24  ; VASK PAST22
ANDNOT C24_SYRE_MED_FORSKYLL  ; ¨
ANDNOT C24_STERILISER  ; PAST22
SET C24_LUT_SYRE  ; PAST22
LD TR0
LD=L(301) MANUELL_KOMMAND &2451410  ; KOMMANDOORD FOR IKKE LINJEKOMMANDOER
%OR C24_VASKEPGM_DRIFT  ; PAST22  FORLOEP INNE
ANDLD
RSET C24_LUT_SYRE  ; PAST22
; rung 6: STERILISERING
LD P_On
OUT TR0
AND=L(301) MANUELL_KOMMAND &1451411  ; KOMMANDOORD FOR IKKE LINJEKOMMANDOER
ANDNOT PGM504_IND_C24  ; VASK PAST22
ANDNOT C24_SYRE_MED_FORSKYLL  ; ¨
ANDNOT C24_LUT_SYRE  ; PAST22
SET C24_STERILISER  ; PAST22
LD TR0
LD=L(301) MANUELL_KOMMAND &2451411  ; KOMMANDOORD FOR IKKE LINJEKOMMANDOER
%OR C24_VASKEPGM_DRIFT  ; PAST22  FORLOEP INNE
ANDLD
RSET C24_STERILISER  ; PAST22

### Section C24_TEMP_OVERVÅKING

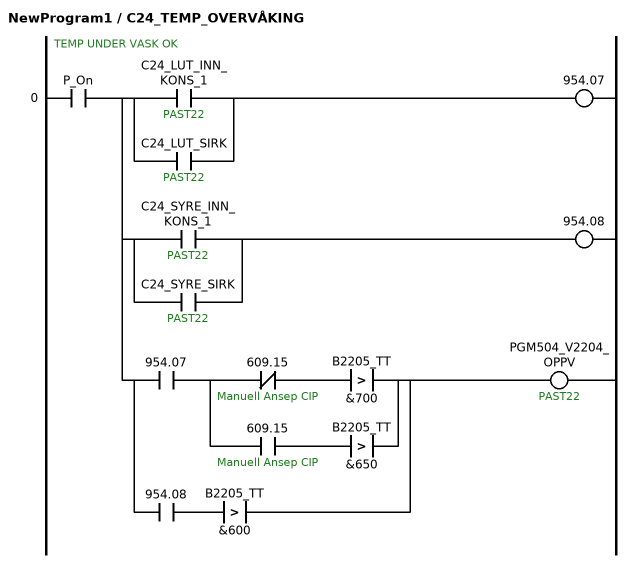
; rung 0: TEMP UNDER VASK OK
LD P_On
OUT TR0
LD C24_LUT_INN_KONS_1  ; PAST22
OR C24_LUT_SIRK  ; PAST22
ANDLD
OUT 954.07
LD TR0
LD C24_SYRE_INN_KONS_1  ; PAST22
OR C24_SYRE_SIRK  ; PAST22
ANDLD
OUT 954.08
LD TR0
LD 954.07
LDNOT 609.15  ; Manuell Ansep CIP
AND>(320) B2205_TT &700
LD 609.15  ; Manuell Ansep CIP
AND>(320) B2205_TT &650
ORLD
ANDLD
LD 954.08
AND>(320) B2205_TT &600
ORLD
ANDLD
OUT PGM504_V2204_OPPV  ; PAST22

### Section VST80_C24_TRINN

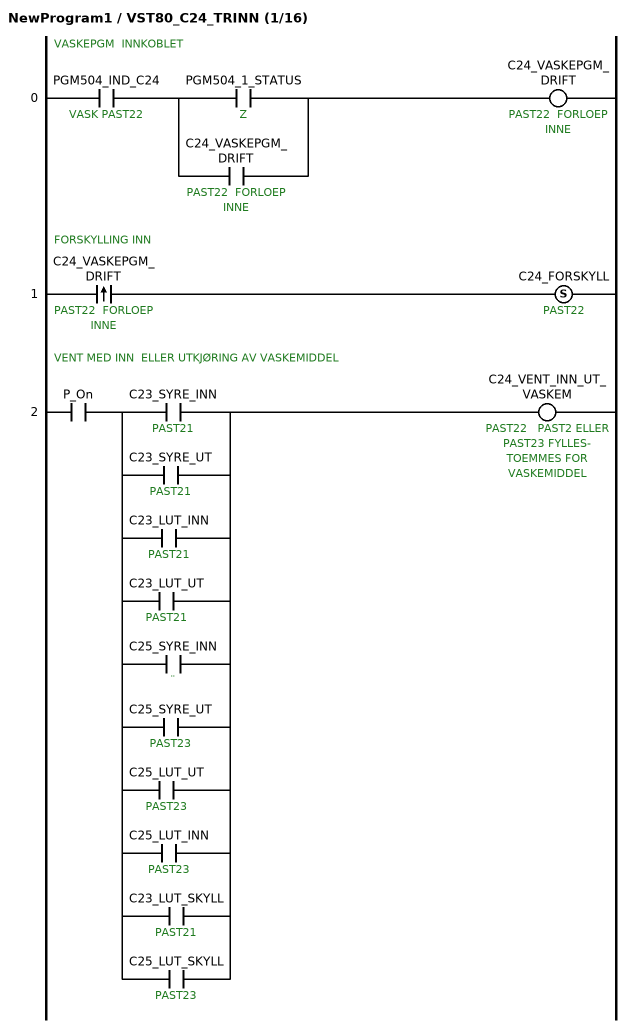
; rung 0: VASKEPGM  INNKOBLET
LD PGM504_IND_C24  ; VASK PAST22
LD PGM504_1_STATUS  ; Z
OR C24_VASKEPGM_DRIFT  ; PAST22  FORLOEP INNE
ANDLD
OUT C24_VASKEPGM_DRIFT  ; PAST22  FORLOEP INNE
; rung 1: FORSKYLLING INN
@LD C24_VASKEPGM_DRIFT  ; PAST22  FORLOEP INNE
SET C24_FORSKYLL  ; PAST22
; rung 2: VENT MED INN  ELLER UTKJØRING AV VASKEMIDDEL
LD P_On
LD C23_SYRE_INN  ; PAST21
OR C23_SYRE_UT  ; PAST21
OR C23_LUT_INN  ; PAST21
OR C23_LUT_UT  ; PAST21
OR C25_SYRE_INN  ; ¨
OR C25_SYRE_UT  ; PAST23
OR C25_LUT_UT  ; PAST23
OR C25_LUT_INN  ; PAST23
OR C23_LUT_SKYLL  ; PAST21
OR C25_LUT_SKYLL  ; PAST23
ANDLD
OUT C24_VENT_INN_UT_VASKEM  ; PAST22   PAST2 ELLER PAST23 FYLLES-TOEMMES FOR VASKEMIDDEL

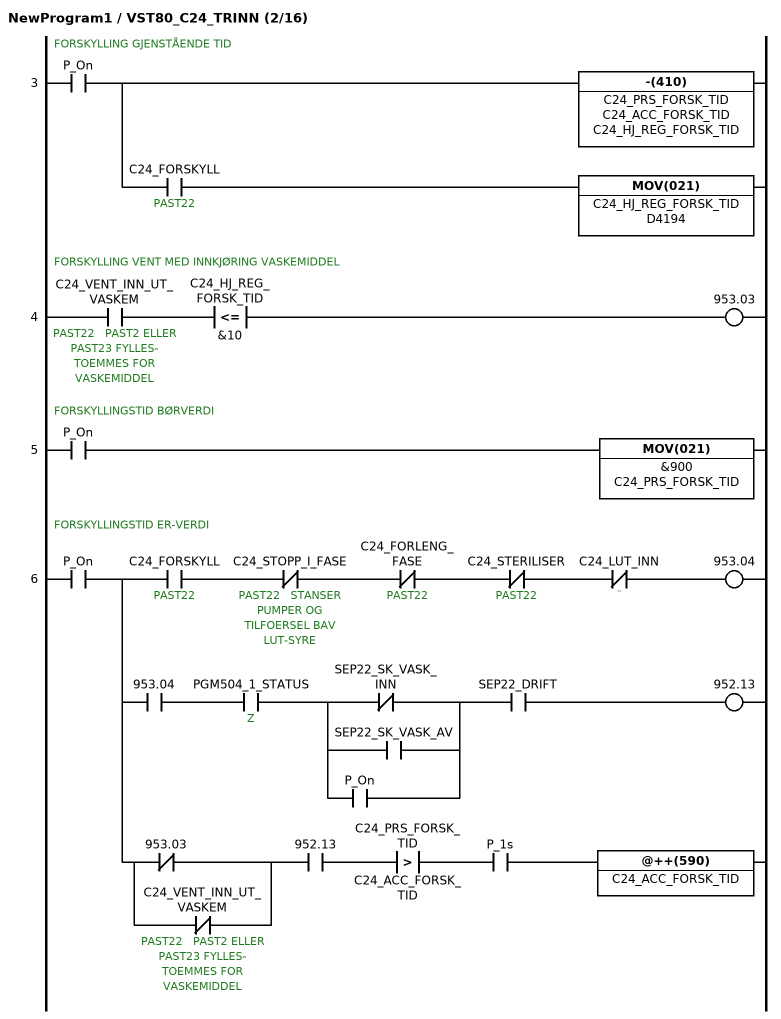
; rung 3: FORSKYLLING GJENSTÅENDE TID
LD P_On
-(410) C24_PRS_FORSK_TID C24_ACC_FORSK_TID C24_HJ_REG_FORSK_TID
AND C24_FORSKYLL  ; PAST22
MOV(021) C24_HJ_REG_FORSK_TID D4194
; rung 4: FORSKYLLING VENT MED INNKJØRING VASKEMIDDEL
LD C24_VENT_INN_UT_VASKEM  ; PAST22   PAST2 ELLER PAST23 FYLLES-TOEMMES FOR VASKEMIDDEL
AND<=(315) C24_HJ_REG_FORSK_TID &10
OUT 953.03
; rung 5: FORSKYLLINGSTID BØRVERDI
LD P_On
MOV(021) &900 C24_PRS_FORSK_TID
; rung 6: FORSKYLLINGSTID ER-VERDI
LD P_On
OUT TR0
AND C24_FORSKYLL  ; PAST22
ANDNOT C24_STOPP_I_FASE  ; PAST22   STANSER PUMPER OG TILFOERSEL BAV LUT-SYRE
ANDNOT C24_FORLENG_FASE  ; PAST22
ANDNOT C24_STERILISER  ; PAST22
ANDNOT C24_LUT_INN  ; ¨
OUT 953.04
LD TR0
AND 953.04
AND PGM504_1_STATUS  ; Z
LDNOT SEP22_SK_VASK_INN
OR SEP22_SK_VASK_AV
OR P_On
ANDLD
AND SEP22_DRIFT
OUT 952.13
LD TR0
LDNOT 953.03
ORNOT C24_VENT_INN_UT_VASKEM  ; PAST22   PAST2 ELLER PAST23 FYLLES-TOEMMES FOR VASKEMIDDEL
ANDLD
AND 952.13
AND>(320) C24_PRS_FORSK_TID C24_ACC_FORSK_TID
AND P_1s
@++(590) C24_ACC_FORSK_TID

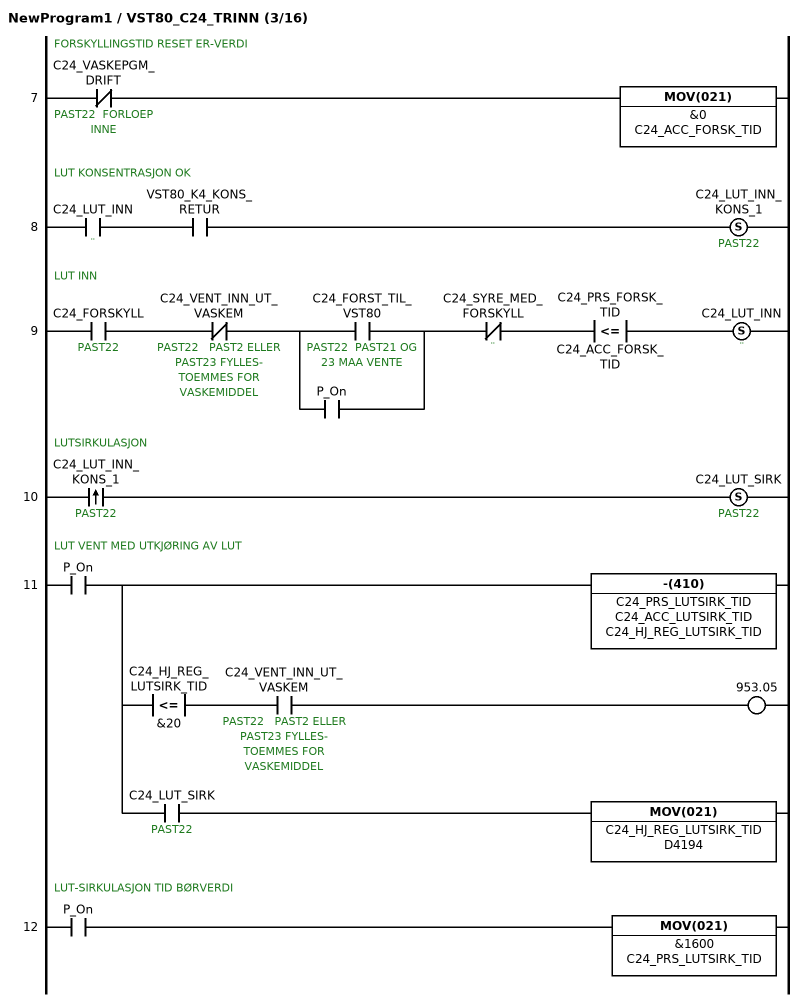
; rung 7: FORSKYLLINGSTID RESET ER-VERDI
LDNOT C24_VASKEPGM_DRIFT  ; PAST22  FORLOEP INNE
MOV(021) &0 C24_ACC_FORSK_TID
; rung 8: LUT KONSENTRASJON OK
LD C24_LUT_INN  ; ¨
AND VST80_K4_KONS_RETUR
SET C24_LUT_INN_KONS_1  ; PAST22
; rung 9: LUT INN
LD C24_FORSKYLL  ; PAST22
ANDNOT C24_VENT_INN_UT_VASKEM  ; PAST22   PAST2 ELLER PAST23 FYLLES-TOEMMES FOR VASKEMIDDEL
LD C24_FORST_TIL_VST80  ; PAST22  PAST21 OG 23 MAA VENTE
OR P_On
ANDLD
ANDNOT C24_SYRE_MED_FORSKYLL  ; ¨
AND<=(315) C24_PRS_FORSK_TID C24_ACC_FORSK_TID
SET C24_LUT_INN  ; ¨
; rung 10: LUTSIRKULASJON
@LD C24_LUT_INN_KONS_1  ; PAST22
SET C24_LUT_SIRK  ; PAST22
; rung 11: LUT VENT MED UTKJØRING AV LUT
LD P_On
OUT TR0
-(410) C24_PRS_LUTSIRK_TID C24_ACC_LUTSIRK_TID C24_HJ_REG_LUTSIRK_TID
AND<=(315) C24_HJ_REG_LUTSIRK_TID &20
AND C24_VENT_INN_UT_VASKEM  ; PAST22   PAST2 ELLER PAST23 FYLLES-TOEMMES FOR VASKEMIDDEL
OUT 953.05
LD TR0
AND C24_LUT_SIRK  ; PAST22
MOV(021) C24_HJ_REG_LUTSIRK_TID D4194
; rung 12: LUT-SIRKULASJON TID BØRVERDI
LD P_On
MOV(021) &1600 C24_PRS_LUTSIRK_TID

